TYPE ref_ele_io :
STRUCT
	param:	ref_ele_param;
	input:	ref_ele_input;
	output:	ref_ele_output;
END_STRUCT
END_TYPE

(* stored: Version 1.1.0.1, ProductVersion 3.1.4024.11
   DUT ref_ele_io: Id {12352ac0-2b67-4d9c-a063-a1297243df14} *)
